TYPE ST_GearAxis :
STRUCT
    nIndex: UINT := 0; //Index of the master axis. 0 means not used
    fRatio: LREAL := 0; //Gearing ratio between master axis and this one
END_STRUCT
END_TYPE

(* stored: Version 1.1.0.1
   DUT ST_GearAxis: Id {dd7a972b-7909-0d2a-2b6a-7781f77a0521} *)
